PROGRAM MAIN
VAR
	fbGetTwinCATVersion	: FB_GetTwinCATVersion;
END_VAR

fbGetTwinCATVersion(sAmsNetId					:= '',
					bExecute					:= TRUE,
					TwinCAT_Major_Version		=>,
					TwinCAT_Minor_Version		=>,
					TwinCAT_Build_Version		=>,
					TwinCAT_Revision_Version	=>,
					sTwinCAT_Version			=>,
					bBusy						=>,
					bError						=>,
					nErrID						=>);

END_PROGRAM

(* stored: Version 1.1.0.1, ProductVersion 3.1.4024.12
   POU MAIN: Id {478a79fb-ccf5-41a4-a3d8-158efc280ff2}, SpecialFunc None *)
